Staubli VAL3: sCenterString.pgx

program sCenterString(string& x_sString, num x_nFillerAsc, num x_nMaxLength)
  local num l_nIndex_i
  local string l_sLeadingSpa
  local string l_sTrailingSpa
begin

  x_sString=left(x_sString,x_nMaxLength)

  //adding spaces to centre the string
  for l_nIndex_i=0 to roundDown((x_nMaxLength-len(x_sString)-1)/2)
    l_sLeadingSpa=l_sLeadingSpa+chr(x_nFillerAsc)
    l_sTrailingSpa=l_sTrailingSpa+chr(x_nFillerAsc)
  endFor

  x_sString=l_sLeadingSpa+x_sString+l_sTrailingSpa

  x_sString=left(x_sString,x_nMaxLength)

end
